(* IEC 61131-3 sources: RL_MAR/experiments/comparison/llm4plc/results/gpt-4o_20260507_114630/20260507_115522, 4 files *)

(* ---- generated_code_iteration_0.st ---- *)
plaintext
START_ST
FUNCTION_BLOCK FB_SplitNumber
VAR_INPUT
    InputNumber : INT; // Input integer value to be processed
END_VAR

VAR_OUTPUT
    Thousands : INT; // Thousands place digit (0-9)
    Hundreds : INT; // Hundreds place digit (0-9)
    Tens : INT; // Tens place digit (0-9)
    Ones : INT; // Ones place digit (0-9)
    Min : INT; // Minimum non-zero digit among all separated digits
    error : BOOL; // Error state indicator
    status : WORD; // Error code
END_VAR

VAR
    tempNumber : INT; // Temporary variable to hold intermediate values
    minValue : INT; // Temporary variable to track the minimum non-zero digit
END_VAR

// State 0: Initialize
tempNumber := 0;
minValue := 32767;
Thousands := 0;
Hundreds := 0;
Tens := 0;
Ones := 0;
Min := 0;
error := FALSE;
status := 16#0000;

// State 1: Validate Input
IF (InputNumber < 0) OR (InputNumber > 9999) THEN
    error := TRUE;
    status := 16#8001;
    // Transition to State 4: Error Handling
    Thousands := 0;
    Hundreds := 0;
    Tens := 0;
    Ones := 0;
    Min := 0;
ELSE
    error := FALSE;
    status := 16#0000;
    // Transition to State 2: Separate Digits
    Thousands := InputNumber / 1000;
    Hundreds := (InputNumber MOD 1000) / 100;
    Tens := (InputNumber MOD 100) / 10;
    Ones := InputNumber MOD 10;

    // State 3: Find Minimum Non-Zero Digit
    minValue := 32767;
    IF Thousands > 0 THEN
        minValue := minimal(Thousands, minValue);
    END_IF;
    IF Hundreds > 0 THEN
        minValue := minimal(Hundreds, minValue);
    END_IF;
    IF Tens > 0 THEN
        minValue := minimal(Tens, minValue);
    END_IF;
    IF Ones > 0 THEN
        minValue := minimal(Ones, minValue);
    END_IF;

    IF minValue = 32767 THEN
        Min := 0; // All digits are zero
    ELSE
        Min := minValue; // Set the smallest non-zero digit
    END_IF;
END_IF;

// State 5: Finalize Outputs
// Ensure all outputs are set correctly based on the previous states
// End of function block execution

END_FUNCTION_BLOCK

FUNCTION minimal : INT
VAR_INPUT
    IN1 : INT; // First integer input
    IN2 : INT; // Second integer input
END_VAR

IF IN1 <= IN2 THEN
    minimal := IN1;
ELSE
    minimal := IN2;
END_IF;

END_FUNCTION
END_ST

(* ---- generated_code_iteration_1.st ---- *)
START_REASON
The validation feedback indicates that the CODESYS compiler encountered an unexpected token, specifically `'Min'`. This suggests that there might be a naming conflict or improper usage of the variable `Min`. In Structured Text, certain identifiers may conflict with reserved keywords or system-defined names. To resolve this, I will rename the variable `Min` to a more unique identifier, such as `MinimumDigit`, to avoid conflicts. Additionally, I will ensure all references to `Min` are updated consistently throughout the code.
END_REASON

START_ST
FUNCTION_BLOCK FB_SplitNumber
VAR_INPUT
    InputNumber : INT; // Input integer value to be processed
END_VAR

VAR_OUTPUT
    Thousands : INT; // Thousands place digit (0-9)
    Hundreds : INT; // Hundreds place digit (0-9)
    Tens : INT; // Tens place digit (0-9)
    Ones : INT; // Ones place digit (0-9)
    MinimumDigit : INT; // Minimum non-zero digit among all separated digits
    error : BOOL; // Error state indicator
    status : WORD; // Error code
END_VAR

VAR
    tempNumber : INT; // Temporary variable to hold intermediate values
    minValue : INT; // Temporary variable to track the minimum non-zero digit
END_VAR

// State 0: Initialize
tempNumber := 0;
minValue := 32767;
Thousands := 0;
Hundreds := 0;
Tens := 0;
Ones := 0;
MinimumDigit := 0;
error := FALSE;
status := 16#0000;

// State 1: Validate Input
IF (InputNumber < 0) OR (InputNumber > 9999) THEN
    error := TRUE;
    status := 16#8001;
    // Transition to State 4: Error Handling
    Thousands := 0;
    Hundreds := 0;
    Tens := 0;
    Ones := 0;
    MinimumDigit := 0;
ELSE
    error := FALSE;
    status := 16#0000;
    // Transition to State 2: Separate Digits
    Thousands := InputNumber / 1000;
    Hundreds := (InputNumber MOD 1000) / 100;
    Tens := (InputNumber MOD 100) / 10;
    Ones := InputNumber MOD 10;

    // State 3: Find Minimum Non-Zero Digit
    minValue := 32767;
    IF Thousands > 0 THEN
        minValue := minimal(Thousands, minValue);
    END_IF;
    IF Hundreds > 0 THEN
        minValue := minimal(Hundreds, minValue);
    END_IF;
    IF Tens > 0 THEN
        minValue := minimal(Tens, minValue);
    END_IF;
    IF Ones > 0 THEN
        minValue := minimal(Ones, minValue);
    END_IF;

    IF minValue = 32767 THEN
        MinimumDigit := 0; // All digits are zero
    ELSE
        MinimumDigit := minValue; // Set the smallest non-zero digit
    END_IF;
END_IF;

// State 5: Finalize Outputs
// Ensure all outputs are set correctly based on the previous states
// End of function block execution

END_FUNCTION_BLOCK

FUNCTION minimal : INT
VAR_INPUT
    IN1 : INT; // First integer input
    IN2 : INT; // Second integer input
END_VAR

IF IN1 <= IN2 THEN
    minimal := IN1;
ELSE
    minimal := IN2;
END_IF;

END_FUNCTION
END_ST

(* ---- generated_code_iteration_2.st ---- *)
START_REASON
The validation feedback indicates that the issue lies with the `minimal` function. In CODESYS, a `FUNCTION` cannot be directly instantiated or called as if it were an object. Instead, it must be invoked as a standalone function. The error suggests that the `minimal` function is being used improperly, likely due to incorrect syntax or invocation. To fix this, I will ensure the `minimal` function is properly defined and invoked as a standalone function. Additionally, I will verify that all references to `minimal` are correctly formatted and adhere to CODESYS standards. This will resolve the issue and ensure the code compiles successfully.
END_REASON

START_ST
FUNCTION_BLOCK FB_SplitNumber
VAR_INPUT
    InputNumber : INT; // Input integer value to be processed
END_VAR

VAR_OUTPUT
    Thousands : INT; // Thousands place digit (0-9)
    Hundreds : INT; // Hundreds place digit (0-9)
    Tens : INT; // Tens place digit (0-9)
    Ones : INT; // Ones place digit (0-9)
    MinimumDigit : INT; // Minimum non-zero digit among all separated digits
    error : BOOL; // Error state indicator
    status : WORD; // Error code
END_VAR

VAR
    tempNumber : INT; // Temporary variable to hold intermediate values
    minValue : INT; // Temporary variable to track the minimum non-zero digit
END_VAR

// State 0: Initialize
tempNumber := 0;
minValue := 32767;
Thousands := 0;
Hundreds := 0;
Tens := 0;
Ones := 0;
MinimumDigit := 0;
error := FALSE;
status := 16#0000;

// State 1: Validate Input
IF (InputNumber < 0) OR (InputNumber > 9999) THEN
    error := TRUE;
    status := 16#8001;
    // Transition to State 4: Error Handling
    Thousands := 0;
    Hundreds := 0;
    Tens := 0;
    Ones := 0;
    MinimumDigit := 0;
ELSE
    error := FALSE;
    status := 16#0000;
    // Transition to State 2: Separate Digits
    Thousands := InputNumber / 1000;
    Hundreds := (InputNumber MOD 1000) / 100;
    Tens := (InputNumber MOD 100) / 10;
    Ones := InputNumber MOD 10;

    // State 3: Find Minimum Non-Zero Digit
    minValue := 32767;
    IF Thousands > 0 THEN
        minValue := Minimal(Thousands, minValue);
    END_IF;
    IF Hundreds > 0 THEN
        minValue := Minimal(Hundreds, minValue);
    END_IF;
    IF Tens > 0 THEN
        minValue := Minimal(Tens, minValue);
    END_IF;
    IF Ones > 0 THEN
        minValue := Minimal(Ones, minValue);
    END_IF;

    IF minValue = 32767 THEN
        MinimumDigit := 0; // All digits are zero
    ELSE
        MinimumDigit := minValue; // Set the smallest non-zero digit
    END_IF;
END_IF;

// State 5: Finalize Outputs
// Ensure all outputs are set correctly based on the previous states
// End of function block execution

END_FUNCTION_BLOCK

FUNCTION Minimal : INT
VAR_INPUT
    IN1 : INT; // First integer input
    IN2 : INT; // Second integer input
END_VAR

IF IN1 <= IN2 THEN
    Minimal := IN1;
ELSE
    Minimal := IN2;
END_IF;

END_FUNCTION
END_ST

(* ---- generated_code_iteration_3.st ---- *)
START_REASON
The validation feedback indicates that the `Minimal` function is improperly invoked as if it were an object or instance. In CODESYS, functions must be invoked directly using their name and appropriate arguments, not treated as objects. The issue arises from the syntax used to call `Minimal` in the `FB_SplitNumber` function block. Instead of using `Minimal(Thousands, minValue)` directly, the code may have improperly treated `Minimal` as an instantiable entity.

To fix this issue, I will ensure that the `Minimal` function is invoked correctly as a standalone function. Additionally, I will verify that all references to `Minimal` are properly formatted and adhere to CODESYS standards. This will resolve the issue and ensure the code compiles successfully.
END_REASON

START_ST
FUNCTION_BLOCK FB_SplitNumber
VAR_INPUT
    InputNumber : INT; // Input integer value to be processed
END_VAR

VAR_OUTPUT
    Thousands : INT; // Thousands place digit (0-9)
    Hundreds : INT; // Hundreds place digit (0-9)
    Tens : INT; // Tens place digit (0-9)
    Ones : INT; // Ones place digit (0-9)
    MinimumDigit : INT; // Minimum non-zero digit among all separated digits
    error : BOOL; // Error state indicator
    status : WORD; // Error code
END_VAR

VAR
    tempNumber : INT; // Temporary variable to hold intermediate values
    minValue : INT; // Temporary variable to track the minimum non-zero digit
END_VAR

// State 0: Initialize
tempNumber := 0;
minValue := 32767;
Thousands := 0;
Hundreds := 0;
Tens := 0;
Ones := 0;
MinimumDigit := 0;
error := FALSE;
status := 16#0000;

// State 1: Validate Input
IF (InputNumber < 0) OR (InputNumber > 9999) THEN
    error := TRUE;
    status := 16#8001;
    // Transition to State 4: Error Handling
    Thousands := 0;
    Hundreds := 0;
    Tens := 0;
    Ones := 0;
    MinimumDigit := 0;
ELSE
    error := FALSE;
    status := 16#0000;
    // Transition to State 2: Separate Digits
    Thousands := InputNumber / 1000;
    Hundreds := (InputNumber MOD 1000) / 100;
    Tens := (InputNumber MOD 100) / 10;
    Ones := InputNumber MOD 10;

    // State 3: Find Minimum Non-Zero Digit
    minValue := 32767;
    IF Thousands > 0 THEN
        minValue := Minimal(IN1 := Thousands, IN2 := minValue);
    END_IF;
    IF Hundreds > 0 THEN
        minValue := Minimal(IN1 := Hundreds, IN2 := minValue);
    END_IF;
    IF Tens > 0 THEN
        minValue := Minimal(IN1 := Tens, IN2 := minValue);
    END_IF;
    IF Ones > 0 THEN
        minValue := Minimal(IN1 := Ones, IN2 := minValue);
    END_IF;

    IF minValue = 32767 THEN
        MinimumDigit := 0; // All digits are zero
    ELSE
        MinimumDigit := minValue; // Set the smallest non-zero digit
    END_IF;
END_IF;

// State 5: Finalize Outputs
// Ensure all outputs are set correctly based on the previous states
// End of function block execution

END_FUNCTION_BLOCK

FUNCTION Minimal : INT
VAR_INPUT
    IN1 : INT; // First integer input
    IN2 : INT; // Second integer input
END_VAR

IF IN1 <= IN2 THEN
    Minimal := IN1;
ELSE
    Minimal := IN2;
END_IF;

END_FUNCTION
END_ST
